// TIA Portal V17 export
// export: Created 2025-03-05T08:03:02.6837359Z, ExportSetting WithDefaults, DisplayName Totally Integrated Automation Portal, DisplayVersion V17 Update 8, DisplayName TIA Portal Openness, DisplayVersion V17 Update 8, DisplayName TIA Portal Version Control Interface, DisplayVersion V17, DisplayName SINAMICS Startdrive Advanced, DisplayVersion V17 SP2, DisplayName SINAMICS Startdrive G110M, G120, G120C, G120D, G120P, G115D, DisplayVersion V17 SP2, DisplayName SINAMICS Startdrive G130, G150, S120, S150, SINAMICS MV, S210, DisplayVersion V17 SP2, DisplayName STEP 7 Professional, DisplayVersion V17 Update 8, DisplayName SINUMERIK ONE STEP 7 Toolbox, DisplayVersion V17 Update 12, DisplayName SINUMERIK 840D sl STEP 7 Toolbox, DisplayVersion V17 Update 12, DisplayName STEP 7 Safety, DisplayVersion V17 Update 6, DisplayName WinCC Advanced, DisplayVersion V17 Update 8
FUNCTION_BLOCK "FB21250_POWDER_ON_OFF_SEQUENCE"   // FB21250, LAD
{ S7_Optimized_Access := 'FALSE' }
VERSION : 0.1
// stored: AutoNumber false, IsIECCheckEnabled false, SetENOAutomatically false, UDAEnableTagReadback false
   VAR_INPUT
      OPTIONS_0 : Byte := 2#0000_0000;   // OPTIONS 0
      REQUEST_INPUT : Bool;   // REQUEST
      GENERAL_CONDITIONS_INPUT : Bool;   // GENERAL CONDITIONS INPUT
      INITIAL_CONDITIONS_INPUT : Bool;   // INITIAL CONDITIONS INPUT
      GAS_FLOW_ACTUAL : Real;   // GAS FLOW ACTUAL
      DISK_SPEED_ACTUAL : Real;   // DISK SPEED ACTUAL
      GAS_SETPOINT : Real;   // GAS SETPOINT
      DISK_SETPOINT : Real;   // DISK SETPOINT
   END_VAR
   VAR_OUTPUT
      DONE : Bool;   // SEQUENCE DONE
   END_VAR
   VAR DB_SPECIFIC
      GENERAL_CONDITIONS : Bool;   // GENERAL CONDITIONS
      INITIAL_CONDITIONS : Bool;   // INITIAL CONDITIONS
      REQUEST_START : Bool;   // REQUEST START
      START_COMMAND : Bool;   // START COMMAND
      RUNNING : Bool := false;   // SEQUENCE RUNNING
      ACTUAL_STEP_GAS : Int := 1;   // ACTUAL STEP GAS
      ACTUAL_STEP_DISK : Int := 1;   // ACTUAL STEP DISK
      MAX_STEPS_GAS : Int := 10;   // MAXIMUM NUMBER OF STEPS FOR GAS
      MAX_STEPS_DISK { ExternalAccessible := 'False'; ExternalVisible := 'False'; ExternalWritable := 'False'} : Int := 10;   // MAXIMUM NUMBER OF STEPS FOR DISK
      GAS_WAIT_STEP : Int;   // GAS PAUSE STEP
      GAS_FLOW_OFFSET { ExternalAccessible := 'False'; ExternalVisible := 'False'; ExternalWritable := 'False'} : Real := 10.0;   // GAS FLOW STEP OFFSET
      DISK_SPEED_OFFSET { ExternalAccessible := 'False'; ExternalVisible := 'False'; ExternalWritable := 'False'} : Real := 10.0;   // DISK SPEED STEP OFFSET
      START_GAS_FLOW { ExternalAccessible := 'False'; ExternalVisible := 'False'; ExternalWritable := 'False'} : Real := 0.0;   // START GAS FLOW
      START_DISK_SPEED : Real := 0.0;   // START DISK SPEED
      GAS_FLOW_MIN : Real := 0.0;   // GAS FLOW MIN
      GAS_FLOW_MAX : Real := 0.0;   // GAS FLOW MAX
      DISK_SPEED_MIN : Real := 0.0;   // DISK SPEED MIN
      DISK_SPEED_MAX : Real := 0.0;   // DISK SPEED MAX
      AUX_SETPOINT_VALUES : Struct
         GAS_FLOW_SETPOINT : Real;   // GAS FLOW SETPOINT
         DISK_SPEED_SETPOINT : Real;   // DISK SPEED SETPOINT
      END_STRUCT;
      STEP_CHANGE_DELAY_GAS : TON_TIME;
      STEP_CHANGE_DELAY_DISK : TON_TIME;
      DONE_DELAY : TON_TIME;
      AUX_1 : Bool;   // AUX PULSE
      AUX_2 : Bool;   // AUX PULSE
      AUX_3 : Bool;   // AUX PULSE
      AUX_4 : Bool;   // AUX PULSE
      AUX_5 : Bool;   // AUX PULSE
   END_VAR
   VAR_TEMP
      DB_NUMBER : DInt;   // DB NUMBER FOR ALARM DECODING
      INPUTS_MASK : Byte;   // INPUTS MASK
      O_BYTE_0 : Struct   // OPTIONS BYTE 0
         ON_SEQUENCE : Bool;   // ON SEQUENCE OPTION
         OFF_SEQUENCE : Bool;   // OFF SEQUENCE OPTION
         SPARE_2 : Bool;
         SPARE_3 : Bool;
         SPARE_4 : Bool;
         SPARE_5 : Bool;
         SPARE_6 : Bool;
         SPARE_7 : Bool;
      END_STRUCT;
   END_VAR
   // STEP_CHANGE_DELAY_GAS.PT := T#200ms;
   // STEP_CHANGE_DELAY_DISK.PT := T#200ms;
   // DONE_DELAY.PT := T#2s;
   VAR_TEMP   // added for the SCL form of the ladder/FBD networks
      _w1 : Bool;
   END_VAR
BEGIN

NETWORK
TITLE = READ INSTANCE DB
      L     DINO;
      +     10#800000;
      T     #DB_NUMBER;


REGION Network 2: OPTIONS
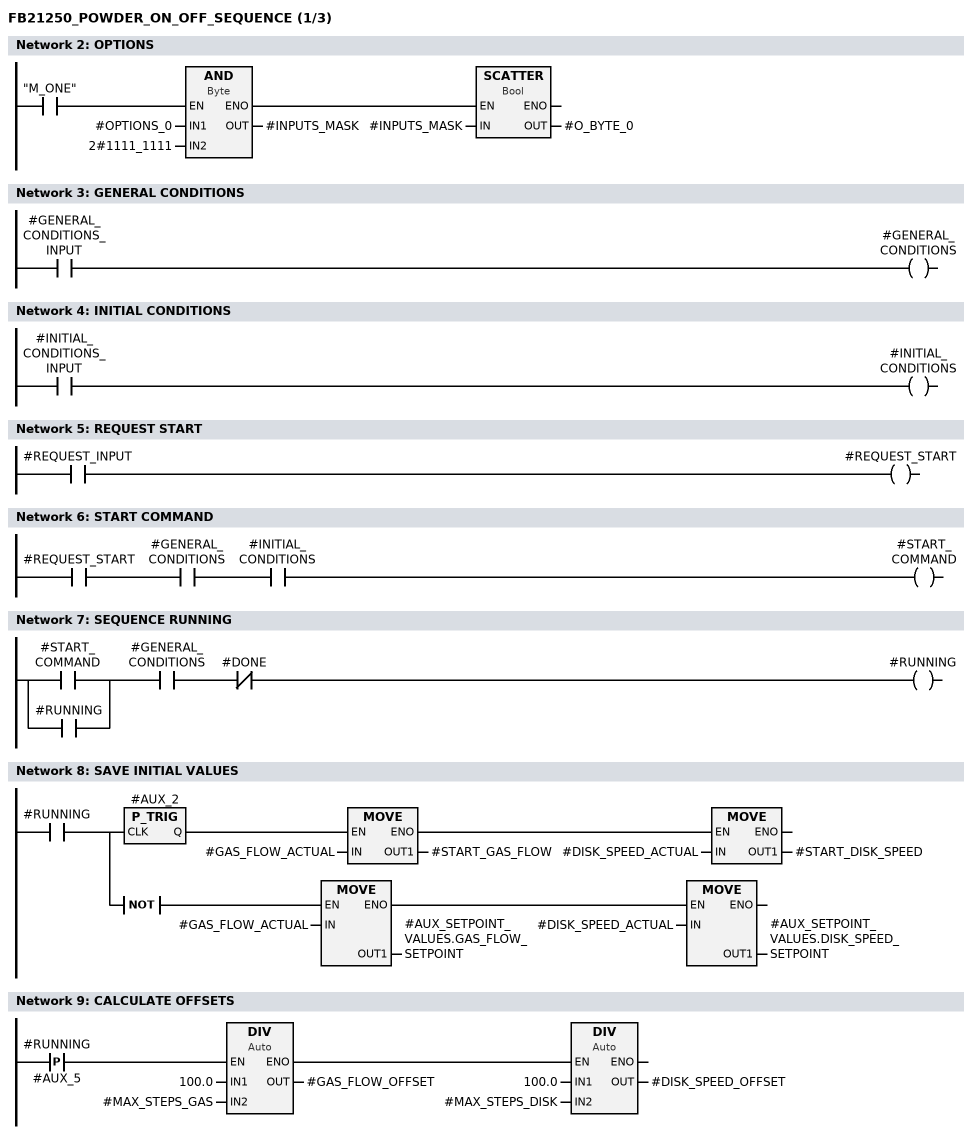
   RUNG wire#powerrail
      Contact( "M_ONE" )
      { S7_Templates := "SrcType := Byte"; S7_GenerateENO := "TRUE" } And(in1 := #OPTIONS_0, in2 := 2#1111_1111, out => #INPUTS_MASK)
      { S7_Templates := "[dest_type := Bool, src_type := Byte]" } SCATTER(IN := #INPUTS_MASK, OUT => #O_BYTE_0)
   END_RUNG
   // the same network as SCL:
   IF "M_ONE" THEN
       #INPUTS_MASK := #OPTIONS_0 AND 2#1111_1111;
       SCATTER(IN := #INPUTS_MASK, OUT => #O_BYTE_0);
   END_IF;
END_REGION

REGION Network 3: GENERAL CONDITIONS
   RUNG wire#powerrail
      Contact( #GENERAL_CONDITIONS_INPUT )
      Coil( #GENERAL_CONDITIONS )
   END_RUNG
   // the same network as SCL:
   #GENERAL_CONDITIONS := #GENERAL_CONDITIONS_INPUT;
END_REGION

REGION Network 4: INITIAL CONDITIONS
   RUNG wire#powerrail
      Contact( #INITIAL_CONDITIONS_INPUT )
      Coil( #INITIAL_CONDITIONS )
   END_RUNG
   // the same network as SCL:
   #INITIAL_CONDITIONS := #INITIAL_CONDITIONS_INPUT;
END_REGION

REGION Network 5: REQUEST START
   RUNG wire#powerrail
      Contact( #REQUEST_INPUT )
      Coil( #REQUEST_START )
   END_RUNG
   // the same network as SCL:
   #REQUEST_START := #REQUEST_INPUT;
END_REGION

REGION Network 6: START COMMAND
   RUNG wire#powerrail
      Contact( #REQUEST_START )
      Contact( #GENERAL_CONDITIONS )
      Contact( #INITIAL_CONDITIONS )
      Coil( #START_COMMAND )
   END_RUNG
   // the same network as SCL:
   #START_COMMAND := #REQUEST_START AND #GENERAL_CONDITIONS AND #INITIAL_CONDITIONS;
END_REGION

REGION Network 7: SEQUENCE RUNNING
   RUNG wire#powerrail
      Contact( #START_COMMAND )
      wire#w1
      Contact( #GENERAL_CONDITIONS )
      I_Contact( #DONE )
      Coil( #RUNNING )
   END_RUNG
   RUNG wire#powerrail
      Contact( #RUNNING )
   END_RUNG wire#w1
   // the same network as SCL:
   #RUNNING := (#START_COMMAND OR #RUNNING) AND #GENERAL_CONDITIONS AND NOT #DONE;
END_REGION

REGION Network 8: SAVE INITIAL VALUES
   RUNG wire#powerrail
      Contact( #RUNNING )
      wire#w1
      P_Trig( #AUX_2 )
      Move(in := #GAS_FLOW_ACTUAL, out1 => #START_GAS_FLOW)
      Move(in := #DISK_SPEED_ACTUAL, out1 => #START_DISK_SPEED)
   END_RUNG
   RUNG wire#w1
      Not()
      Move(in := #GAS_FLOW_ACTUAL, out1 => #AUX_SETPOINT_VALUES.GAS_FLOW_SETPOINT)
      Move(in := #DISK_SPEED_ACTUAL, out1 => #AUX_SETPOINT_VALUES.DISK_SPEED_SETPOINT)
   END_RUNG
   // the same network as SCL:
   #_w1 := #RUNNING AND NOT #AUX_2;   // rising edge
   #AUX_2 := #RUNNING;
   IF #_w1 THEN
       #START_GAS_FLOW := #GAS_FLOW_ACTUAL;
       #START_DISK_SPEED := #DISK_SPEED_ACTUAL;
   END_IF;
   IF NOT #RUNNING THEN
       #AUX_SETPOINT_VALUES.GAS_FLOW_SETPOINT := #GAS_FLOW_ACTUAL;
       #AUX_SETPOINT_VALUES.DISK_SPEED_SETPOINT := #DISK_SPEED_ACTUAL;
   END_IF;
END_REGION

REGION Network 9: CALCULATE OFFSETS
   RUNG wire#powerrail
      P_Contact(operand := #RUNNING, bit := #AUX_5)
      Div(in1 := 100.0, in2 := #MAX_STEPS_GAS, out => #GAS_FLOW_OFFSET)
      Div(in1 := 100.0, in2 := #MAX_STEPS_DISK, out => #DISK_SPEED_OFFSET)
   END_RUNG
   // the same network as SCL:
   #_w1 := #RUNNING AND NOT #AUX_5;   // rising edge of #RUNNING
   #AUX_5 := #RUNNING;
   IF #_w1 THEN
       #GAS_FLOW_OFFSET := 100.0 / #MAX_STEPS_GAS;
       #DISK_SPEED_OFFSET := 100.0 / #MAX_STEPS_DISK;
   END_IF;
END_REGION

REGION Network 10: CALCULATE VALUES DISK
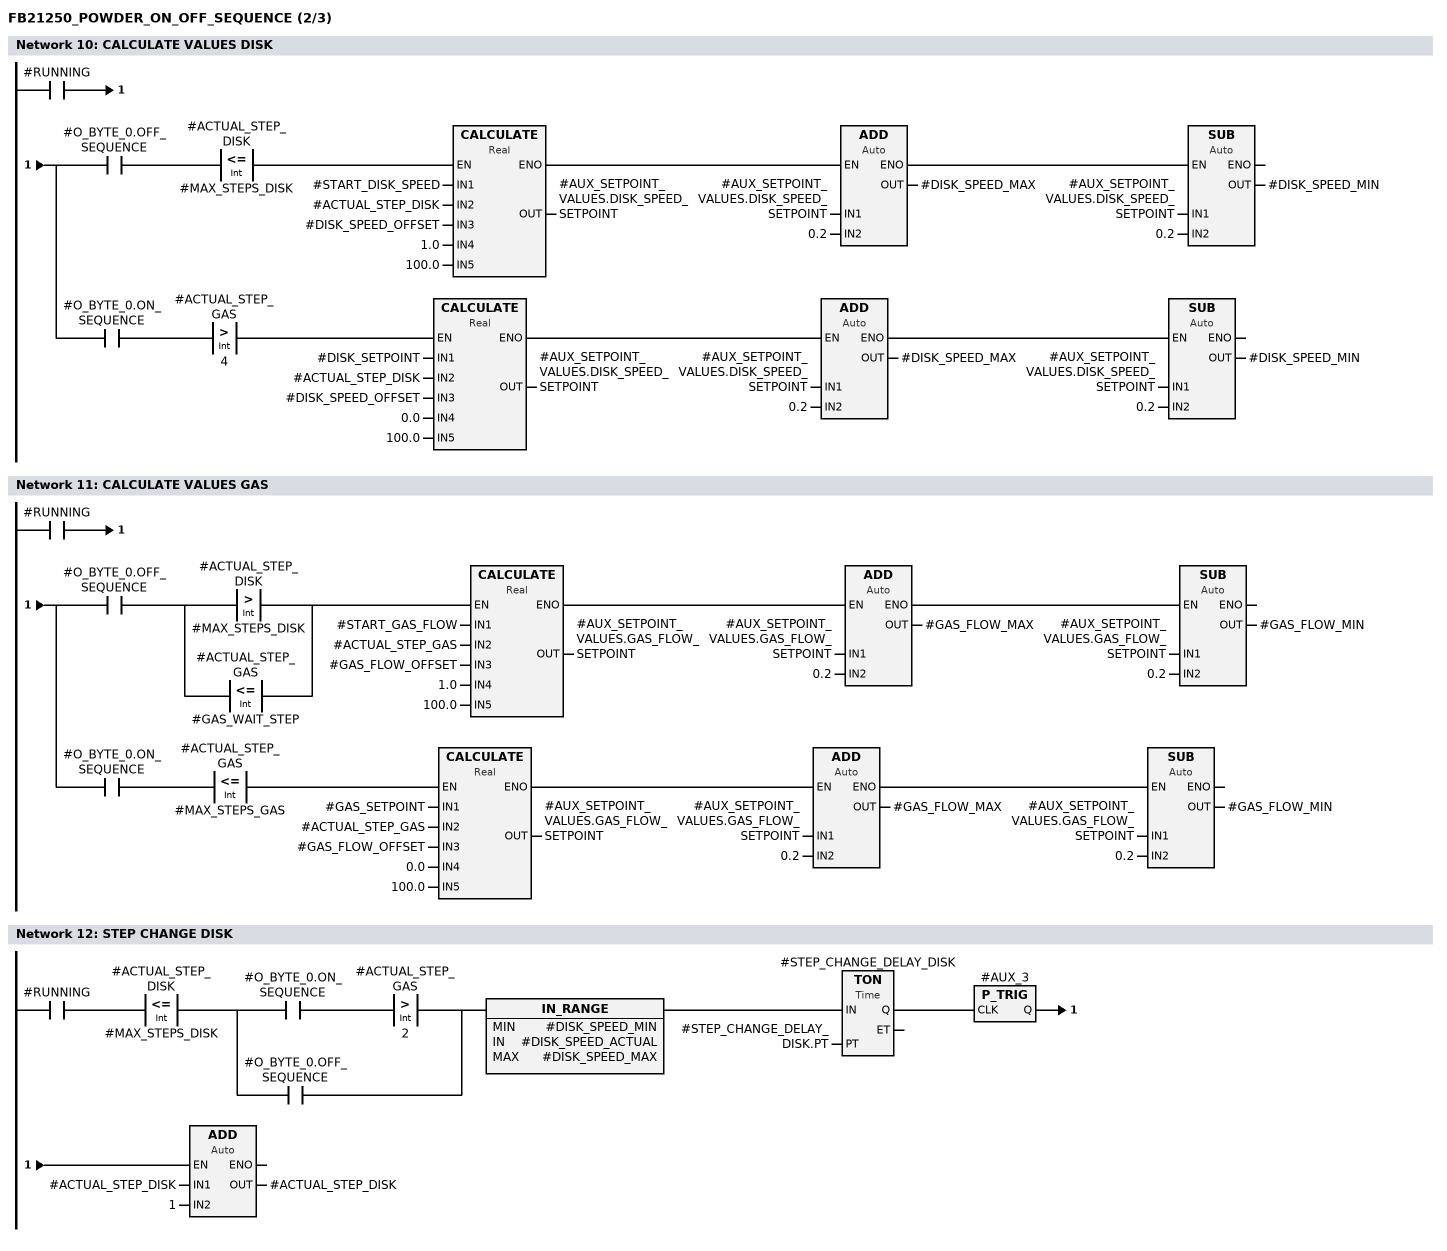
   RUNG wire#powerrail
      Contact( #RUNNING )
      wire#w1
      Contact( #O_BYTE_0.OFF_SEQUENCE )
      { S7_Templates := "SrcType := Int" } LE_Contact(in1 := #ACTUAL_STEP_DISK, in2 := #MAX_STEPS_DISK)
      { S7_Templates := "SrcType := Real"; S7_Expression := "(IN1)*(IN4-(IN2*(IN3/IN5)))" } Calculate(in1 := #START_DISK_SPEED, in2 := #ACTUAL_STEP_DISK, in3 := #DISK_SPEED_OFFSET, in4 := 1.0, in5 := 100.0, out => #AUX_SETPOINT_VALUES.DISK_SPEED_SETPOINT)
      Add(in1 := #AUX_SETPOINT_VALUES.DISK_SPEED_SETPOINT, in2 := 0.2, out => #DISK_SPEED_MAX)
      Sub(in1 := #AUX_SETPOINT_VALUES.DISK_SPEED_SETPOINT, in2 := 0.2, out => #DISK_SPEED_MIN)
   END_RUNG
   RUNG wire#w1
      Contact( #O_BYTE_0.ON_SEQUENCE )
      { S7_Templates := "SrcType := Int" } GT_Contact(in1 := #ACTUAL_STEP_GAS, in2 := 4)
      { S7_Templates := "SrcType := Real"; S7_Expression := "(IN1)*(IN4+(IN2*(IN3/IN5)))" } Calculate(in1 := #DISK_SETPOINT, in2 := #ACTUAL_STEP_DISK, in3 := #DISK_SPEED_OFFSET, in4 := 0.0, in5 := 100.0, out => #AUX_SETPOINT_VALUES.DISK_SPEED_SETPOINT)
      Add(in1 := #AUX_SETPOINT_VALUES.DISK_SPEED_SETPOINT, in2 := 0.2, out => #DISK_SPEED_MAX)
      Sub(in1 := #AUX_SETPOINT_VALUES.DISK_SPEED_SETPOINT, in2 := 0.2, out => #DISK_SPEED_MIN)
   END_RUNG
   // the same network as SCL:
   IF #RUNNING AND #O_BYTE_0.OFF_SEQUENCE AND (#ACTUAL_STEP_DISK <= #MAX_STEPS_DISK) THEN
       #AUX_SETPOINT_VALUES.DISK_SPEED_SETPOINT := (#START_DISK_SPEED)*(1.0-(#ACTUAL_STEP_DISK*(#DISK_SPEED_OFFSET/100.0)));
       #DISK_SPEED_MAX := #AUX_SETPOINT_VALUES.DISK_SPEED_SETPOINT + 0.2;
       #DISK_SPEED_MIN := #AUX_SETPOINT_VALUES.DISK_SPEED_SETPOINT - 0.2;
   END_IF;
   IF #RUNNING AND #O_BYTE_0.ON_SEQUENCE AND (#ACTUAL_STEP_GAS > 4) THEN
       #AUX_SETPOINT_VALUES.DISK_SPEED_SETPOINT := (#DISK_SETPOINT)*(0.0+(#ACTUAL_STEP_DISK*(#DISK_SPEED_OFFSET/100.0)));
       #DISK_SPEED_MAX := #AUX_SETPOINT_VALUES.DISK_SPEED_SETPOINT + 0.2;
       #DISK_SPEED_MIN := #AUX_SETPOINT_VALUES.DISK_SPEED_SETPOINT - 0.2;
   END_IF;
END_REGION

REGION Network 11: CALCULATE VALUES GAS
   RUNG wire#powerrail
      Contact( #RUNNING )
      wire#w1
      Contact( #O_BYTE_0.OFF_SEQUENCE )
      wire#w2
      { S7_Templates := "SrcType := Int" } GT_Contact(in1 := #ACTUAL_STEP_DISK, in2 := #MAX_STEPS_DISK)
      wire#w3
      { S7_Templates := "SrcType := Real"; S7_Expression := "(IN1)*(IN4-(IN2*(IN3/IN5)))" } Calculate(in1 := #START_GAS_FLOW, in2 := #ACTUAL_STEP_GAS, in3 := #GAS_FLOW_OFFSET, in4 := 1.0, in5 := 100.0, out => #AUX_SETPOINT_VALUES.GAS_FLOW_SETPOINT)
      Add(in1 := #AUX_SETPOINT_VALUES.GAS_FLOW_SETPOINT, in2 := 0.2, out => #GAS_FLOW_MAX)
      Sub(in1 := #AUX_SETPOINT_VALUES.GAS_FLOW_SETPOINT, in2 := 0.2, out => #GAS_FLOW_MIN)
   END_RUNG
   RUNG wire#w2
      { S7_Templates := "SrcType := Int" } LE_Contact(in1 := #ACTUAL_STEP_GAS, in2 := #GAS_WAIT_STEP)
   END_RUNG wire#w3
   RUNG wire#w1
      Contact( #O_BYTE_0.ON_SEQUENCE )
      { S7_Templates := "SrcType := Int" } LE_Contact(in1 := #ACTUAL_STEP_GAS, in2 := #MAX_STEPS_GAS)
      { S7_Templates := "SrcType := Real"; S7_Expression := "(IN1)*(IN4+(IN2*(IN3/IN5)))" } Calculate(in1 := #GAS_SETPOINT, in2 := #ACTUAL_STEP_GAS, in3 := #GAS_FLOW_OFFSET, in4 := 0.0, in5 := 100.0, out => #AUX_SETPOINT_VALUES.GAS_FLOW_SETPOINT)
      Add(in1 := #AUX_SETPOINT_VALUES.GAS_FLOW_SETPOINT, in2 := 0.2, out => #GAS_FLOW_MAX)
      Sub(in1 := #AUX_SETPOINT_VALUES.GAS_FLOW_SETPOINT, in2 := 0.2, out => #GAS_FLOW_MIN)
   END_RUNG
   // the same network as SCL:
   IF #RUNNING AND #O_BYTE_0.OFF_SEQUENCE AND ((#ACTUAL_STEP_DISK > #MAX_STEPS_DISK) OR (#ACTUAL_STEP_GAS <= #GAS_WAIT_STEP)) THEN
       #AUX_SETPOINT_VALUES.GAS_FLOW_SETPOINT := (#START_GAS_FLOW)*(1.0-(#ACTUAL_STEP_GAS*(#GAS_FLOW_OFFSET/100.0)));
       #GAS_FLOW_MAX := #AUX_SETPOINT_VALUES.GAS_FLOW_SETPOINT + 0.2;
       #GAS_FLOW_MIN := #AUX_SETPOINT_VALUES.GAS_FLOW_SETPOINT - 0.2;
   END_IF;
   IF #RUNNING AND #O_BYTE_0.ON_SEQUENCE AND (#ACTUAL_STEP_GAS <= #MAX_STEPS_GAS) THEN
       #AUX_SETPOINT_VALUES.GAS_FLOW_SETPOINT := (#GAS_SETPOINT)*(0.0+(#ACTUAL_STEP_GAS*(#GAS_FLOW_OFFSET/100.0)));
       #GAS_FLOW_MAX := #AUX_SETPOINT_VALUES.GAS_FLOW_SETPOINT + 0.2;
       #GAS_FLOW_MIN := #AUX_SETPOINT_VALUES.GAS_FLOW_SETPOINT - 0.2;
   END_IF;
END_REGION

REGION Network 12: STEP CHANGE DISK
   RUNG wire#powerrail
      Contact( #RUNNING )
      { S7_Templates := "SrcType := Int" } LE_Contact(in1 := #ACTUAL_STEP_DISK, in2 := #MAX_STEPS_DISK)
      wire#w1
      Contact( #O_BYTE_0.ON_SEQUENCE )
      { S7_Templates := "SrcType := Int" } GT_Contact(in1 := #ACTUAL_STEP_GAS, in2 := 2)
      wire#w2
      { S7_Templates := "SrcType := Real" } InRange(min := #DISK_SPEED_MIN, in := #DISK_SPEED_ACTUAL, max := #DISK_SPEED_MAX)
      { S7_Templates := "time_type := Time" } #STEP_CHANGE_DELAY_DISK.TON(pt := #STEP_CHANGE_DELAY_DISK.PT, et =>)
      P_Trig( #AUX_3 )
      Add(in1 := #ACTUAL_STEP_DISK, in2 := 1, out => #ACTUAL_STEP_DISK)
   END_RUNG
   RUNG wire#w1
      Contact( #O_BYTE_0.OFF_SEQUENCE )
   END_RUNG wire#w2
   // the same network as SCL:
   #STEP_CHANGE_DELAY_DISK(IN := #RUNNING AND (#ACTUAL_STEP_DISK <= #MAX_STEPS_DISK) AND ((#O_BYTE_0.ON_SEQUENCE AND (#ACTUAL_STEP_GAS > 2)) OR #O_BYTE_0.OFF_SEQUENCE) AND (#DISK_SPEED_MIN <= #DISK_SPEED_ACTUAL) AND (#DISK_SPEED_ACTUAL <= #DISK_SPEED_MAX),   // TON
                           PT := #STEP_CHANGE_DELAY_DISK.PT);
   #_w1 := #STEP_CHANGE_DELAY_DISK.Q AND NOT #AUX_3;   // rising edge
   #AUX_3 := #STEP_CHANGE_DELAY_DISK.Q;
   IF #_w1 THEN #ACTUAL_STEP_DISK := #ACTUAL_STEP_DISK + 1; END_IF;
END_REGION

REGION Network 13: STEP CHANGE GAS
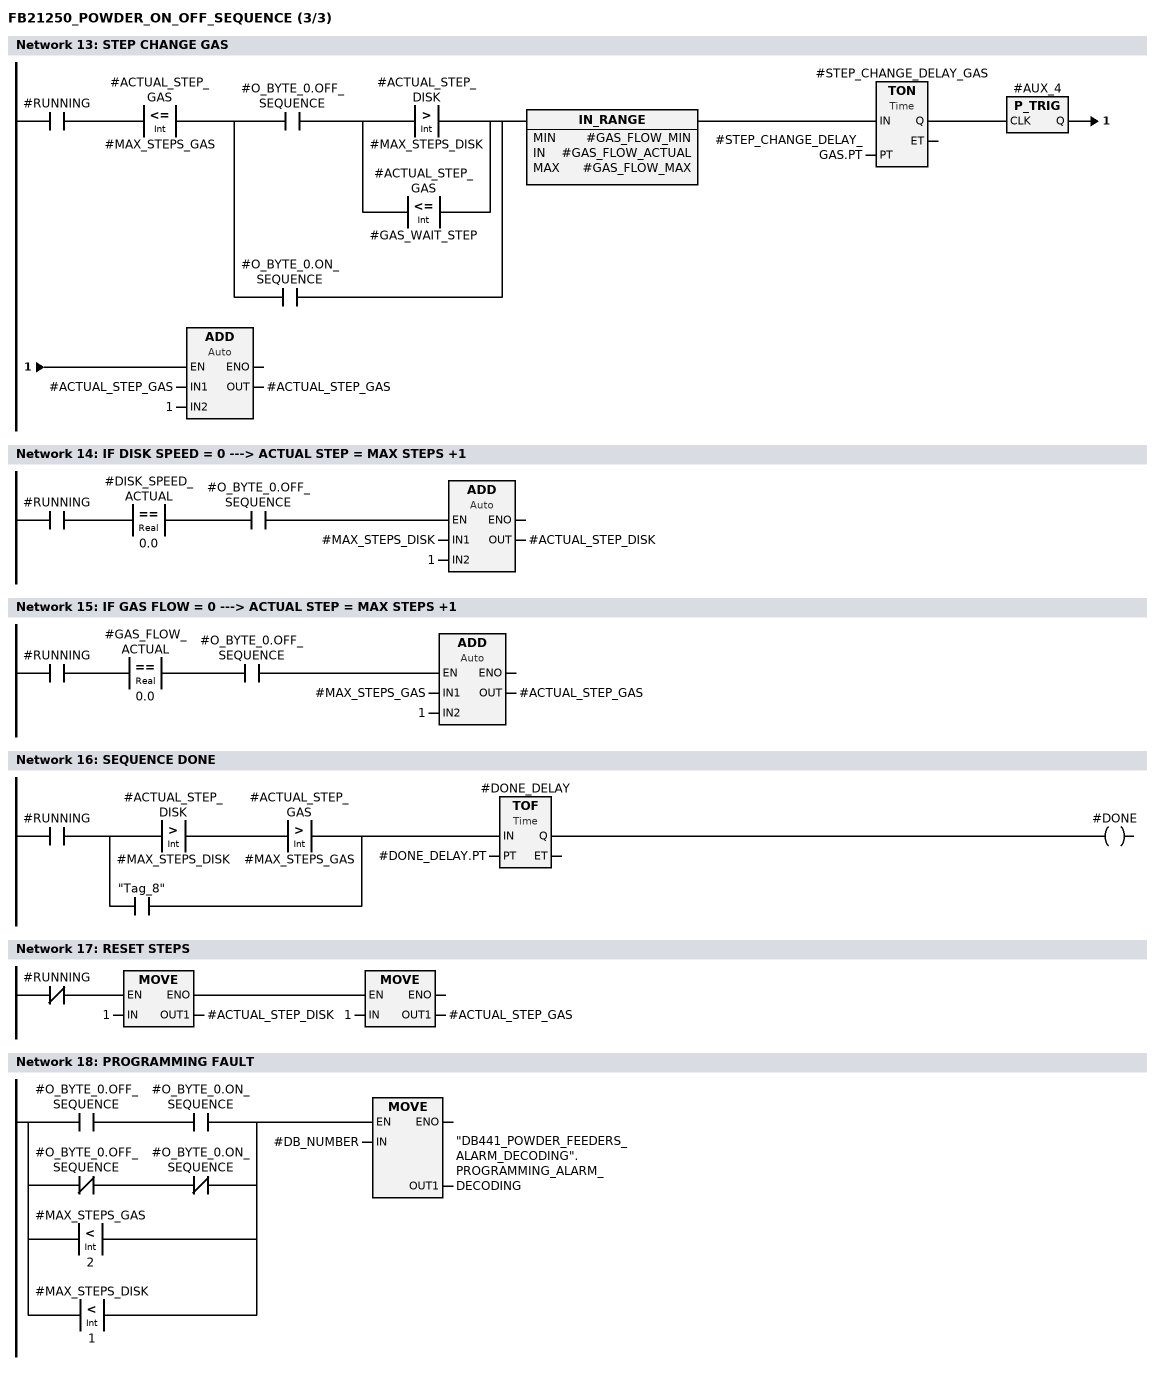
   RUNG wire#powerrail
      Contact( #RUNNING )
      { S7_Templates := "SrcType := Int" } LE_Contact(in1 := #ACTUAL_STEP_GAS, in2 := #MAX_STEPS_GAS)
      wire#w1
      Contact( #O_BYTE_0.OFF_SEQUENCE )
      wire#w2
      { S7_Templates := "SrcType := Int" } GT_Contact(in1 := #ACTUAL_STEP_DISK, in2 := #MAX_STEPS_DISK)
      wire#w3
      { S7_Templates := "SrcType := Real" } InRange(min := #GAS_FLOW_MIN, in := #GAS_FLOW_ACTUAL, max := #GAS_FLOW_MAX)
      { S7_Templates := "time_type := Time" } #STEP_CHANGE_DELAY_GAS.TON(pt := #STEP_CHANGE_DELAY_GAS.PT, et =>)
      P_Trig( #AUX_4 )
      Add(in1 := #ACTUAL_STEP_GAS, in2 := 1, out => #ACTUAL_STEP_GAS)
   END_RUNG
   RUNG wire#w2
      { S7_Templates := "SrcType := Int" } LE_Contact(in1 := #ACTUAL_STEP_GAS, in2 := #GAS_WAIT_STEP)
   END_RUNG wire#w3
   RUNG wire#w1
      Contact( #O_BYTE_0.ON_SEQUENCE )
   END_RUNG wire#w3
   // the same network as SCL:
   #STEP_CHANGE_DELAY_GAS(IN := #RUNNING AND (#ACTUAL_STEP_GAS <= #MAX_STEPS_GAS) AND ((#O_BYTE_0.OFF_SEQUENCE AND ((#ACTUAL_STEP_DISK > #MAX_STEPS_DISK) OR (#ACTUAL_STEP_GAS <= #GAS_WAIT_STEP))) OR #O_BYTE_0.ON_SEQUENCE) AND (#GAS_FLOW_MIN <= #GAS_FLOW_ACTUAL) AND (#GAS_FLOW_ACTUAL <= #GAS_FLOW_MAX),   // TON
                          PT := #STEP_CHANGE_DELAY_GAS.PT);
   #_w1 := #STEP_CHANGE_DELAY_GAS.Q AND NOT #AUX_4;   // rising edge
   #AUX_4 := #STEP_CHANGE_DELAY_GAS.Q;
   IF #_w1 THEN #ACTUAL_STEP_GAS := #ACTUAL_STEP_GAS + 1; END_IF;
END_REGION

REGION Network 14: IF DISK SPEED = 0 ---> ACTUAL STEP = MAX STEPS +1
   RUNG wire#powerrail
      Contact( #RUNNING )
      { S7_Templates := "SrcType := Real" } EQ_Contact(in1 := #DISK_SPEED_ACTUAL, in2 := 0.0)
      Contact( #O_BYTE_0.OFF_SEQUENCE )
      Add(in1 := #MAX_STEPS_DISK, in2 := 1, out => #ACTUAL_STEP_DISK)
   END_RUNG
   // the same network as SCL:
   IF #RUNNING AND (#DISK_SPEED_ACTUAL = 0.0) AND #O_BYTE_0.OFF_SEQUENCE THEN
       #ACTUAL_STEP_DISK := #MAX_STEPS_DISK + 1;
   END_IF;
END_REGION

REGION Network 15: IF GAS FLOW = 0 ---> ACTUAL STEP = MAX STEPS +1
   RUNG wire#powerrail
      Contact( #RUNNING )
      { S7_Templates := "SrcType := Real" } EQ_Contact(in1 := #GAS_FLOW_ACTUAL, in2 := 0.0)
      Contact( #O_BYTE_0.OFF_SEQUENCE )
      Add(in1 := #MAX_STEPS_GAS, in2 := 1, out => #ACTUAL_STEP_GAS)
   END_RUNG
   // the same network as SCL:
   IF #RUNNING AND (#GAS_FLOW_ACTUAL = 0.0) AND #O_BYTE_0.OFF_SEQUENCE THEN
       #ACTUAL_STEP_GAS := #MAX_STEPS_GAS + 1;
   END_IF;
END_REGION

REGION Network 16: SEQUENCE DONE
   RUNG wire#powerrail
      Contact( #RUNNING )
      wire#w1
      { S7_Templates := "SrcType := Int" } GT_Contact(in1 := #ACTUAL_STEP_DISK, in2 := #MAX_STEPS_DISK)
      { S7_Templates := "SrcType := Int" } GT_Contact(in1 := #ACTUAL_STEP_GAS, in2 := #MAX_STEPS_GAS)
      wire#w2
      { S7_Templates := "time_type := Time" } #DONE_DELAY.TOF(pt := #DONE_DELAY.PT, et =>)
      Coil( #DONE )
   END_RUNG
   RUNG wire#w1
      Contact( "Tag_8" )
   END_RUNG wire#w2
   // the same network as SCL:
   #DONE_DELAY(IN := #RUNNING AND (((#ACTUAL_STEP_DISK > #MAX_STEPS_DISK) AND (#ACTUAL_STEP_GAS > #MAX_STEPS_GAS)) OR "Tag_8"),   // TOF
               PT := #DONE_DELAY.PT);
   #DONE := #DONE_DELAY.Q;
END_REGION

REGION Network 17: RESET STEPS
   RUNG wire#powerrail
      I_Contact( #RUNNING )
      Move(in := 1, out1 => #ACTUAL_STEP_DISK)
      Move(in := 1, out1 => #ACTUAL_STEP_GAS)
   END_RUNG
   // the same network as SCL:
   IF NOT #RUNNING THEN
       #ACTUAL_STEP_DISK := 1;
       #ACTUAL_STEP_GAS := 1;
   END_IF;
END_REGION

REGION Network 18: PROGRAMMING FAULT
   RUNG wire#powerrail
      Contact( #O_BYTE_0.OFF_SEQUENCE )
      Contact( #O_BYTE_0.ON_SEQUENCE )
      wire#w1
      Move(in := #DB_NUMBER, out1 => "DB441_POWDER_FEEDERS_ALARM_DECODING".PROGRAMMING_ALARM_DECODING)
   END_RUNG
   RUNG wire#powerrail
      I_Contact( #O_BYTE_0.OFF_SEQUENCE )
      I_Contact( #O_BYTE_0.ON_SEQUENCE )
   END_RUNG wire#w1
   RUNG wire#powerrail
      { S7_Templates := "SrcType := Int" } LT_Contact(in1 := #MAX_STEPS_GAS, in2 := 2)
   END_RUNG wire#w1
   RUNG wire#powerrail
      { S7_Templates := "SrcType := Int" } LT_Contact(in1 := #MAX_STEPS_DISK, in2 := 1)
   END_RUNG wire#w1
   // the same network as SCL:
   IF (#O_BYTE_0.OFF_SEQUENCE AND #O_BYTE_0.ON_SEQUENCE) OR (NOT #O_BYTE_0.OFF_SEQUENCE AND NOT #O_BYTE_0.ON_SEQUENCE) OR (#MAX_STEPS_GAS < 2) OR (#MAX_STEPS_DISK < 1) THEN
       "DB441_POWDER_FEEDERS_ALARM_DECODING".PROGRAMMING_ALARM_DECODING := #DB_NUMBER;
   END_IF;
END_REGION
END_FUNCTION_BLOCK
